{attribute 'qualified_only'}
{attribute 'strict'}
TYPE Colors :
(
	Red,
	Green,
	Orange,
	Yellow
);
END_TYPE

(* stored: Version 1.1.0.1, ProductVersion 3.1.4024.11
   DUT Colors: Id {24708ed7-468f-47cf-8c04-d4e7572a9ae7} *)
